// TIA Portal V20 export
DATA_BLOCK "InterfaceSignals"   // DB196
// stored: MemoryReserve 100
   VAR
      HMI_Interface_Mode : Bool;
      "Button Value" : Array[0..99] of "LER_SignalsInput";
   END_VAR
BEGIN
END_DATA_BLOCK
